// Mitsubishi GX Works2 project: Count_time01   PLC: Q02/Q02H

PROGRAM MAIN
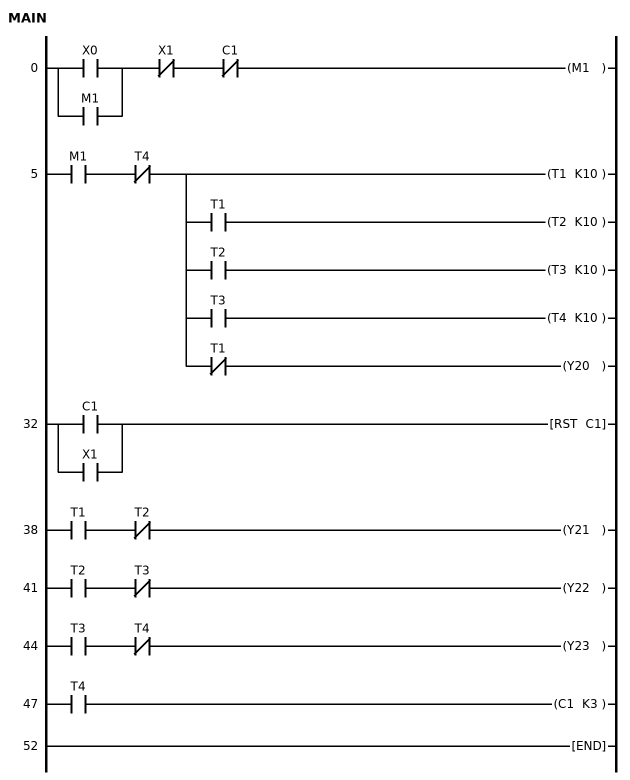
0     LD      X0
      OR      M1
      ANI     X1
      ANI     C1
      OUT     M1
5     LD      M1
      ANI     T4
      OUT     T1 K10
      MPS
      AND     T1
      OUT     T2 K10
      MRD
      AND     T2
      OUT     T3 K10
      MRD
      AND     T3
      OUT     T4 K10
      MPP
      ANI     T1
      OUT     Y20
32    LD      C1
      OR      X1
      RST     C1
38    LD      T1
      ANI     T2
      OUT     Y21
41    LD      T2
      ANI     T3
      OUT     Y22
44    LD      T3
      ANI     T4
      OUT     Y23
47    LD      T4
      OUT     C1 K3
52    END
END_PROGRAM
